// TIA Portal V17 export
// export: Created 2023-02-14T02:49:35.9135343Z, ExportSetting WithDefaults, DisplayName Totally Integrated Automation Portal, DisplayVersion V17, DisplayName TIA Portal Openness, DisplayVersion V17, DisplayName TIA Portal Teamcenter Gateway, DisplayVersion V17, DisplayName TIA Portal Version Control Interface, DisplayVersion V17, DisplayName SINAMICS Startdrive Advanced, DisplayVersion V17, DisplayName SINAMICS Startdrive G130, G150, S120, S150, SINAMICS MV, S210, DisplayVersion V17, DisplayName SINAMICS Startdrive G110M, G120, G120C, G120D, G120P, G115D, DisplayVersion V17, DisplayName STEP 7 Professional, DisplayVersion V17, DisplayName STEP 7 Safety, DisplayVersion V17, DisplayName WinCC Professional, DisplayVersion V17
DATA_BLOCK "IO_Valve_T01_HWT"   // DB301
VERSION : 0.1
// stored: AutoNumber false, DBAccessibleFromOPCUA true, DBAccessibleFromWebserver true, InstanceOfName IO Valve T01 HWT, InstanceOfType FB
"IO Valve T01 HWT"
   // VAR_INPUT
   //    lock : Bool;
   //    Init : Bool;
   //    Reset : Bool;
   // END_VAR
   // VAR
   //    "AV-01.01" { S7_SetPoint := 'True'} : "Valve";
   //    "AV-01.02" { S7_SetPoint := 'True'} : "Valve";
   //    "AV-01.03" { S7_SetPoint := 'True'} : "Valve";
   //    "AV-01.04" { S7_SetPoint := 'True'} : "Valve";
   //    "AV-01.05" { S7_SetPoint := 'True'} : "Valve";
   //    "AV-01.06" { S7_SetPoint := 'True'} : "Valve";
   //    "AV-01.07" { S7_SetPoint := 'True'} : "Valve";
   //    "AV-01.08" { S7_SetPoint := 'True'} : "Valve";
   //    "AV-01.09" { S7_SetPoint := 'True'} : "Valve";
   //    "AV-01.10" { S7_SetPoint := 'True'} : "Valve";
   //    "AV-01.11" { S7_SetPoint := 'True'} : "Valve";
   //    "AV-01.12" { S7_SetPoint := 'True'} : "Valve";
   //    "AV-01.13" { S7_SetPoint := 'True'} : "Valve";
   //    "AV-01.14" { S7_SetPoint := 'True'} : "Valve";
   //    "AV-01.15" { S7_SetPoint := 'True'} : "Valve";
   //    "CV-01.01" { S7_SetPoint := 'True'} : "Valve";
   // END_VAR
BEGIN
END_DATA_BLOCK
